FUNCTION_BLOCK FB_TrafficLight
VAR
    state : INT;  // 0=Red, 1=RedAmber, 2=Green, 3=Amber
END_VAR

METHOD Step : INT
CASE state OF
    0:
        state := 1;
    1:
        state := 2;
    2:
        state := 0;
    3:
        state := 0;
END_CASE;
Step := state;
END_METHOD

END_FUNCTION_BLOCK

(* stored: Version 1.1.0.1
   POU FB_TrafficLight: Id {bb714433-311f-4a1c-a08f-af4230b2ee6c}, SpecialFunc None
   Method Step: Id {4122d60d-9b9b-4f5d-bbcb-8cf5fc27f0fb} *)
